{attribute 'GeneratedUsingTerminal: EK1100-0000-0018'}
{attribute addProperty BoxType "EK1100-0000-0018"}
{attribute addProperty Id "Term_24_EL1809EL1809_32157CFD20Term_25_EL2809EL2809_2B6483BD19"}
{attribute addProperty CRC "74331346"}
{attribute addProperty Size "39"}
{attribute addProperty Name "Term 23 (EK1100)"}
TYPE Term_23_EK1100_046E34D2 EXTENDS EK1100_1FC0878B :
STRUCT
	{attribute addProperty Name "Term 24 (EL1809)"}
	{attribute addProperty PreviousPort "Term 23 (EK1100) : B"}
	Term_24_EL1809 : EL1809_32157CFD;
	{attribute addProperty Name "Term 25 (EL2809)"}
	{attribute addProperty PreviousPort "Term 24 (EL1809) : B"}
	Term_25_EL2809 : EL2809_2B6483BD;
END_STRUCT
END_TYPE

(* stored: Version 1.2.0.0, ProductVersion 3.1.4024.11
   DUT Term_23_EK1100_046E34D2: Id {247054ae-0967-0488-1e4d-dded7760690f} *)
